PROGRAM tuning
VAR
END_VAR

END_PROGRAM

(* stored: Version 1.1.0.1, ProductVersion 3.1.4024.4
   POU tuning: Id {e720b919-2168-4ef5-8c08-ecf23986856b}, SpecialFunc None *)
